Staubli VAL3: OnF8.pgx

program OnF8(string x_sMsg)
  local num l_i
  local string l_sYesNo[2]
begin
  //
  l_sYesNo[0]="是"
  l_sYesNo[1]="否"
  call user:questionDialog(x_sMsg,l_sYesNo,l_i)
  if l_i==0 or l_i==1
    bExit=true
    cls()
  endIf
  bUserRefresh=true
end
